(* IEC 61131-3 sources: LStream-JSON-XML/src/Timer, 2 files *)

(* ---- ITimerFunction.st ---- *)
NAMESPACE Simatic.Ax.Timer

    INTERFACE PUBLIC ITimerFunctions
        METHOD TimerFunction : BOOL
            VAR_INPUT
                signal : BOOL;
                duration : LTIME;
            END_VAR
        END_METHOD
    END_INTERFACE

END_NAMESPACE

(* ---- TimerFunctionImpl.st ---- *)
USING System.Timer;

NAMESPACE Simatic.Ax.Timer

    CLASS PUBLIC TimerFunctionsImpl IMPLEMENTS ITimerFunctions
        VAR
            Timer : OnDelay;
        END_VAR

        METHOD PUBLIC TimerFunction : BOOL
            VAR_INPUT
                signal : BOOL;
                duration : LTIME;
            END_VAR

            Timer(signal := signal, duration := duration);
            TimerFunction := Timer.output;

        END_METHOD
    END_CLASS

END_NAMESPACE
